DATA_BLOCK "Test"
{ S7_Optimized_Access := 'TRUE' }
VERSION : 0.1
NON_RETAIN
   VAR
      Member : Struct
         Member1 : Struct
            Member2 : Struct
               Membe3 : Struct
                  Member4 : Bool;
               END_STRUCT;
            END_STRUCT;
         END_STRUCT;
      END_STRUCT;
   END_VAR


BEGIN

END_DATA_BLOCK

